FUNCTION_BLOCK SludgeBufferLogic (* Composite Function Block Type *)
  (* Standard: 61499-2 *)
  (* Version 0.0, 10/24/2023, SESA685388, Schneider Electric, template *)
  PACKAGE SE.Nereda;
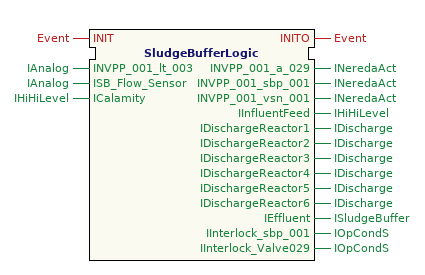
  EVENT_INPUT
    INIT; (* Initialization Request *)
  END_EVENT
  EVENT_OUTPUT
    INITO; (* Initialization Confirm *)
  END_EVENT
  SOCKETS
    INVPP_001_lt_003 : IAnalog;
    ISB_Flow_Sensor : IAnalog;
    ICalamity : IHiHiLevel;
  END_SOCKETS
  PLUGS
    INVPP_001_a_029 : INeredaAct;
    INVPP_001_sbp_001 : INeredaAct;
    INVPP_001_vsn_001 : INeredaAct;
    IInfluentFeed : IHiHiLevel;
    IDischargeReactor1 : IDischarge;
    IDischargeReactor2 : IDischarge;
    IDischargeReactor3 : IDischarge;
    IDischargeReactor4 : IDischarge;
    IDischargeReactor5 : IDischarge;
    IDischargeReactor6 : IDischarge;
    IEffluent : ISludgeBuffer;
  END_PLUGS
  PLUGS
    IInterlock_sbp_001 : IOpCondS; (* Condition summary chain output to downstream block *)
    IInterlock_Valve029 : IOpCondS; (* Condition summary chain output to downstream block *)
  END_PLUGS
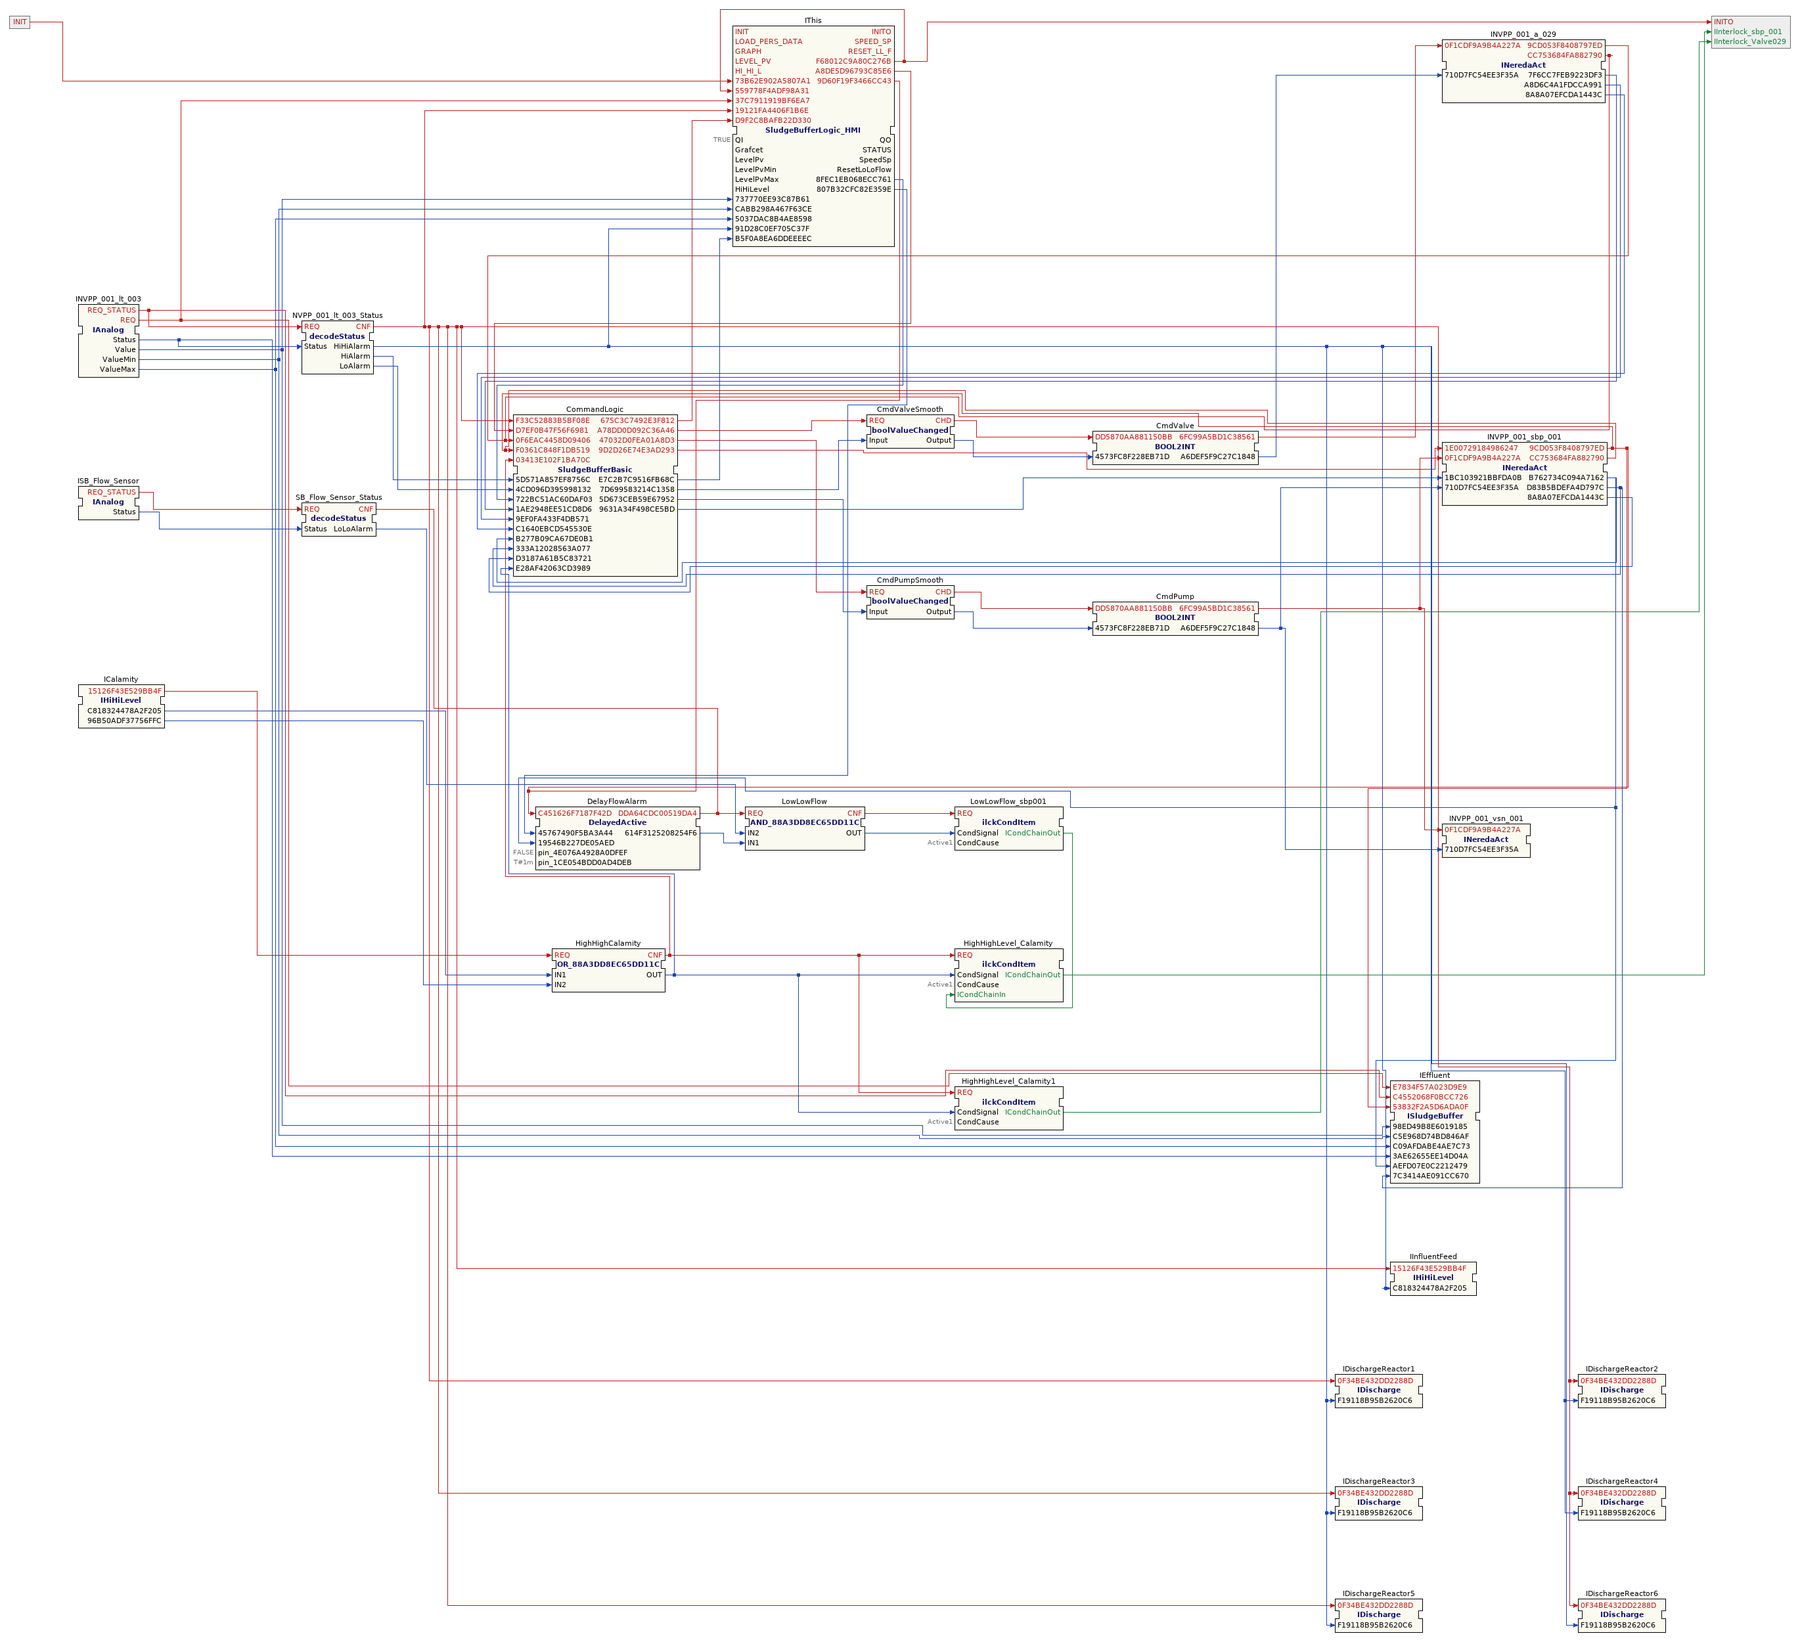
  (* 01 - FUNCTIONNAL INPUT INTERFACE *)
  (* 00 - INITIALIZATION *)
  (* 05 - LOGIC *)
  (* 06 - HMI INTERFACE *)
  (* CommandLogic *)
  (* 02 - FUNCTIONNAL OUTPUT INTERFACE *)
  (* Interlock *)
  (* 03 - FIELD INTERFACE *)
  FBS
    CmdValveSmooth : boolValueChanged;
    CmdPumpSmooth : boolValueChanged;
    IThis : SludgeBufferLogic_HMI(QI := TRUE);
    NVPP_001_lt_003_Status : decodeStatus; {SET_ATTRIBUTE(Configuration.Component.HideUnusedPorts, )}
    SB_Flow_Sensor_Status : decodeStatus; {SET_ATTRIBUTE(Configuration.Component.HideUnusedPorts, )}
    CommandLogic : SludgeBufferBasic;
    DelayFlowAlarm : DelayedActive(pin_4E076A4928A0DFEF := FALSE, pin_1CE054BDD0AD4DEB := T#1m);
    LowLowFlow : AND_88A3DD8EC65DD11C; {SET_ATTRIBUTE(Configuration.GenericFBType.InterfaceParams, Runtime.Standard#CNT:=2;OUT:BOOL)}
    LowLowFlow_sbp001 : ilckCondItem(CondCause := Active1);
    HighHighLevel_Calamity : ilckCondItem(CondCause := Active1);
    HighHighCalamity : OR_88A3DD8EC65DD11C; {SET_ATTRIBUTE(Configuration.GenericFBType.InterfaceParams, Runtime.Standard#CNT:=2;OUT:BOOL)}
    CmdValve : BOOL2INT;
    CmdPump : BOOL2INT;
    HighHighLevel_Calamity1 : ilckCondItem(CondCause := Active1);
  END_FBS
  EVENT_CONNECTIONS
    INVPP_001_lt_003.REQ_STATUS TO NVPP_001_lt_003_Status.REQ;
    ISB_Flow_Sensor.REQ_STATUS TO SB_Flow_Sensor_Status.REQ;
    HighHighCalamity.CNF TO HighHighLevel_Calamity.REQ;
    LowLowFlow.CNF TO LowLowFlow_sbp001.REQ;
    SB_Flow_Sensor_Status.CNF TO LowLowFlow.REQ;
    INIT TO IThis.73B62E902A5807A1;
    IThis.F68012C9A80C276B TO IThis.559778F4ADF98A31;
    INVPP_001_lt_003.REQ TO IThis.37C7911919BF6EA7;
    IThis.F68012C9A80C276B TO INITO;
    NVPP_001_lt_003_Status.CNF TO IThis.19121FA4406F1B6E;
    NVPP_001_lt_003_Status.CNF TO IDischargeReactor1.0F34BE432DD2288D;
    NVPP_001_lt_003_Status.CNF TO IDischargeReactor2.0F34BE432DD2288D;
    NVPP_001_lt_003_Status.CNF TO IDischargeReactor3.0F34BE432DD2288D;
    NVPP_001_lt_003_Status.CNF TO IDischargeReactor4.0F34BE432DD2288D;
    NVPP_001_lt_003_Status.CNF TO IDischargeReactor5.0F34BE432DD2288D;
    NVPP_001_lt_003_Status.CNF TO IDischargeReactor6.0F34BE432DD2288D;
    NVPP_001_lt_003_Status.CNF TO IInfluentFeed.15126F43E529BB4F;
    NVPP_001_lt_003_Status.CNF TO CommandLogic.F33C52883B5BF08E;
    ICalamity.15126F43E529BB4F TO HighHighCalamity.REQ;
    CommandLogic.675C3C7492E3F812 TO IThis.D9F2C8BAFB22D330;
    IThis.A8DE5D96793C85E6 TO CommandLogic.D7EF0B47F56F6981;
    IThis.9D60F19F3466CC43 TO DelayFlowAlarm.C451626F7187F42D;
    INVPP_001_a_029.9CD053F8408797ED TO CommandLogic.0F6EAC4458D09406;
    INVPP_001_a_029.CC753684FA882790 TO CommandLogic.0F6EAC4458D09406;
    INVPP_001_sbp_001.9CD053F8408797ED TO CommandLogic.F0361C848F1DB519;
    INVPP_001_sbp_001.CC753684FA882790 TO CommandLogic.F0361C848F1DB519;
    HighHighCalamity.CNF TO CommandLogic.03413E102F1BA70C;
    CommandLogic.A78DD0D092C36A46 TO CmdValveSmooth.REQ;
    CommandLogic.47032D0FEA01A8D3 TO CmdPumpSmooth.REQ;
    CommandLogic.9D2D26E74E3AD293 TO INVPP_001_sbp_001.1E00729184986247;
    CmdValveSmooth.CHD TO CmdValve.DD5870AA881150BB;
    CmdPumpSmooth.CHD TO CmdPump.DD5870AA881150BB;
    CmdValve.6FC99A5BD1C38561 TO INVPP_001_a_029.0F1CDF9A9B4A227A;
    CmdPump.6FC99A5BD1C38561 TO INVPP_001_sbp_001.0F1CDF9A9B4A227A;
    CmdPump.6FC99A5BD1C38561 TO INVPP_001_vsn_001.0F1CDF9A9B4A227A;
    INVPP_001_sbp_001.9CD053F8408797ED TO DelayFlowAlarm.C451626F7187F42D;
    DelayFlowAlarm.DDA64CDC00519DA4 TO LowLowFlow.REQ;
    INVPP_001_lt_003.REQ TO IEffluent.E7834F57A023D9E9;
    INVPP_001_lt_003.REQ_STATUS TO IEffluent.C4552068F0BCC726;
    INVPP_001_sbp_001.9CD053F8408797ED TO IEffluent.53832F2A5D6ADA0F;
    HighHighCalamity.CNF TO HighHighLevel_Calamity1.REQ;
  END_CONNECTIONS
  DATA_CONNECTIONS
    INVPP_001_lt_003.Status TO NVPP_001_lt_003_Status.Status;
    ISB_Flow_Sensor.Status TO SB_Flow_Sensor_Status.Status;
    HighHighCalamity.OUT TO HighHighLevel_Calamity.CondSignal;
    LowLowFlow.OUT TO LowLowFlow_sbp001.CondSignal;
    SB_Flow_Sensor_Status.LoLoAlarm TO LowLowFlow.IN2;
    INVPP_001_lt_003.Value TO IThis.737770EE93C87B61;
    INVPP_001_lt_003.ValueMin TO IThis.CABB298A467F63CE;
    INVPP_001_lt_003.ValueMax TO IThis.5037DAC8B4AE8598;
    NVPP_001_lt_003_Status.HiHiAlarm TO IThis.91D28C0EF705C37F;
    NVPP_001_lt_003_Status.HiHiAlarm TO IInfluentFeed.C818324478A2F205;
    NVPP_001_lt_003_Status.HiHiAlarm TO IDischargeReactor1.F19118B95B2620C6;
    NVPP_001_lt_003_Status.HiHiAlarm TO IDischargeReactor2.F19118B95B2620C6;
    NVPP_001_lt_003_Status.HiHiAlarm TO IDischargeReactor3.F19118B95B2620C6;
    NVPP_001_lt_003_Status.HiHiAlarm TO IDischargeReactor4.F19118B95B2620C6;
    NVPP_001_lt_003_Status.HiHiAlarm TO IDischargeReactor5.F19118B95B2620C6;
    NVPP_001_lt_003_Status.HiHiAlarm TO IDischargeReactor6.F19118B95B2620C6;
    NVPP_001_lt_003_Status.HiAlarm TO CommandLogic.5D571A857EF8756C;
    NVPP_001_lt_003_Status.LoAlarm TO CommandLogic.4CD096D395998132;
    ICalamity.C818324478A2F205 TO HighHighCalamity.IN1;
    ICalamity.96B50ADF37756FFC TO HighHighCalamity.IN2;
    CommandLogic.E7C2B7C9516FB68C TO IThis.B5F0A8EA6DDEEEEC;
    IThis.8FEC1EB068ECC761 TO CommandLogic.722BC51AC60DAF03;
    IThis.807B32CFC82E359E TO DelayFlowAlarm.45767490F5BA3A44;
    INVPP_001_a_029.7F6CC7FEB9223DF3 TO CommandLogic.1AE2948EE51CD8D6;
    INVPP_001_a_029.A8D6C4A1FDCCA991 TO CommandLogic.9EF0FA433F4DB571;
    INVPP_001_a_029.8A8A07EFCDA1443C TO CommandLogic.C1640EBCD545530E;
    INVPP_001_sbp_001.B762734C094A7162 TO CommandLogic.B277B09CA67DE0B1;
    INVPP_001_sbp_001.D83B5BDEFA4D797C TO CommandLogic.333A12028563A077;
    INVPP_001_sbp_001.8A8A07EFCDA1443C TO CommandLogic.D3187A61B5C83721;
    HighHighCalamity.OUT TO CommandLogic.E28AF42063CD3989;
    CommandLogic.7D699583214C1358 TO CmdValveSmooth.Input;
    CommandLogic.5D673CEB59E67952 TO CmdPumpSmooth.Input;
    CommandLogic.9631A34F498CE5BD TO INVPP_001_sbp_001.1BC103921BBFDA0B;
    CmdValveSmooth.Output TO CmdValve.4573FC8F228EB71D;
    CmdPumpSmooth.Output TO CmdPump.4573FC8F228EB71D;
    CmdValve.A6DEF5F9C27C1848 TO INVPP_001_a_029.710D7FC54EE3F35A;
    CmdPump.A6DEF5F9C27C1848 TO INVPP_001_sbp_001.710D7FC54EE3F35A;
    CmdPump.A6DEF5F9C27C1848 TO INVPP_001_vsn_001.710D7FC54EE3F35A;
    INVPP_001_sbp_001.B762734C094A7162 TO DelayFlowAlarm.19546B227DE05AED;
    DelayFlowAlarm.614F3125208254F6 TO LowLowFlow.IN1;
    INVPP_001_lt_003.Value TO IEffluent.98ED49B8E6019185;
    INVPP_001_lt_003.ValueMin TO IEffluent.C5E968D74BD846AF;
    INVPP_001_lt_003.ValueMax TO IEffluent.C09AFDABE4AE7C73;
    INVPP_001_lt_003.Status TO IEffluent.3AE62655EE14D04A;
    INVPP_001_sbp_001.B762734C094A7162 TO IEffluent.AEFD07E0C2212479;
    INVPP_001_sbp_001.D83B5BDEFA4D797C TO IEffluent.7C3414AE091CC670;
    HighHighCalamity.OUT TO HighHighLevel_Calamity1.CondSignal;
  END_CONNECTIONS
  ADAPTER_CONNECTIONS
    LowLowFlow_sbp001.ICondChainOut TO HighHighLevel_Calamity.ICondChainIn;
    HighHighLevel_Calamity.ICondChainOut TO IInterlock_sbp_001;
    HighHighLevel_Calamity1.ICondChainOut TO IInterlock_Valve029;
  END_CONNECTIONS
END_FUNCTION_BLOCK
